PROGRAM StringHelper
VAR
END_VAR

METHOD EndsWith : BOOL
VAR_INPUT
	str		: Tc2_System.T_MaxString;
	char	: T_Char;	
END_VAR
EndsWith := Tc2_Standard.RIGHT(str, 1) = char;
END_METHOD

// Checks if the sourceString contains the stringToFind string. 
// Size of the source string is only limited to TwinCAT limitaitons, which in theory is not limited.
// Returns TRUE if found, else FALSE. Position of the found strimg is provided in the "position" output variable.
METHOD FindStringWithin : BOOL
VAR_INPUT
	sourceString	: ANY;	// String to look at
	stringToFind	: Tc2_System.T_MaxString; // String that should be containted in the sourceString
END_VAR
VAR_OUTPUT
	position	: DINT;	// Position of the found string
END_VAR

VAR
	tmpStr						: POINTER TO Tc2_System.T_MaxString;
	charIndex					: DINT;
	currentMatchingCharIndex	: DINT;
	tmpByte						: POINTER TO BYTE;
	firstCharPosition 			: dint;
END_VAR
IF NOT F_DoesVarTypeEqual(sourceString, IBaseLibrary.TYPE_STRING) THEN
	RETURN;
END_IF

IF sourceString.diSize <= SIZEOF(Tc2_System.T_MaxString) THEN
	tmpStr := __NEW(BYTE, SIZEOF(Tc2_System.T_MaxString));
	Tc2_System.MEMCPY(
		destAddr := tmpStr,
		srcAddr := sourceString.pValue,
		n := DINT_TO_UDINT(sourceString.diSize));
	//tmpStr := sourceString.pValue;
	position :=  Tc2_Standard.FIND(tmpStr^, stringToFind);
	FindStringWithin := position <> 0;
	__DELETE(tmpStr);
	RETURN;
END_IF

FOR charIndex := 0 TO sourceString.diSize BY 1 DO
	
	// Byte wise comparison, if matching byte, start filling the compared string
	tmpByte := sourceString.pValue + charIndex * SIZEOF(BYTE);
	// For debug purpose
	tmpStr := tmpByte;
	IF tmpbyte^ = stringToFind[currentMatchingCharIndex] THEN
		IF firstCharPosition = 0 THEN
			firstCharPosition := charIndex + 1;
		END_IF
		currentMatchingCharIndex := currentMatchingCharIndex + 1;
	ELSE
		currentMatchingCharIndex := 0;
		firstCharPosition := 0;
	END_IF
	
	// When index = str lenght - 1, we have found the entire string, exit the loop.
	IF currentMatchingCharIndex = (Tc2_Standard.LEN(stringToFind)) THEN
		position := firstCharPosition;
		FindStringWithin := TRUE;
		EXIT;
	END_IF
END_FOR
END_METHOD

// Joins the provided string with the string to add.
// The refStr is altered in the process, this no additional assignments are required as oposed to CONCAT which returns the resulting string.
METHOD Join
VAR_INPUT
	refStr		: REFERENCE TO Tc2_System.T_MaxString;
	strToJoin	: Tc2_System.T_MaxString;
END_VAR
refStr := Tc2_Standard.CONCAT(refStr, strToJoin);
END_METHOD

// Checks if STRING `str` starts with the `char`
// Returs TRUE if first character in the provided string is `char` provided
METHOD StartsWith : BOOL
VAR_INPUT
	str		: Tc2_System.T_MaxString;	// String to be checked
	char	: T_Char;	// Character that the string will be checked, if it starts with it.
END_VAR
StartsWith := Tc2_System.F_ToCHR(str[0]) = char;
END_METHOD

// Converts the provided string to all lower case and returns the converted value.
METHOD ToLowerCase : T_MaxString
VAR_INPUT
	str	: Tc2_System.T_MaxString;	// Source string
END_VAR
ToLowerCase := Tc2_Utilities.F_ToLCase(in := str);
END_METHOD

// Converts the input string to all lower case. Size of the string is irrelevant
METHOD ToLowerCase_UnlimitedSize
VAR_INPUT
	str	: ANY;
END_VAR

VAR
	charIndex	: DINT;
	ptrChar		: POINTER TO T_Char;
	char		: T_Char;
	malloc		: FB_Malloc(0,0);
	ptrByte		: POINTER TO BYTE;
END_VAR
IF NOT F_DoesVarTypeEqual(str, IBaseLibrary.TYPE_STRING) THEN
	RETURN;
END_IF

malloc.Allocate(1, str.diSize - 1);		
FOR charIndex := 0 TO str.diSize - 1 BY 1 DO
	ptrChar := str.pValue + DINT_TO_DWORD(charIndex);
	char := ToLowerCase(ptrChar^);
	ptrByte := ADR(char);
	malloc.Set(charIndex, ptrByte^);
END_FOR

Tc2_System.MEMCPY(
	destAddr := str.pValue, 
	srcAddr := malloc.Properties.StartAddress, 
	n := DINT_TO_UDINT(str.diSize - 1));
	
malloc.Free();
END_METHOD

// Converts the provided string to all upper case and returns the converted value.
METHOD ToUpperCase : Tc2_System.T_MaxString
VAR_INPUT
	str	: Tc2_System.T_MaxString;	// Source string
END_VAR
ToUpperCase := Tc2_Utilities.F_ToUCase(in := str);
END_METHOD

METHOD ToUpperCase_UnlimitedSize
VAR_INPUT
	str	: ANY;
END_VAR	

VAR
	charIndex	: DINT;
	ptrChar		: POINTER TO T_Char;
	char		: T_Char;
	malloc		: FB_Malloc(0,0);
	ptrByte		: POINTER TO BYTE;
END_VAR
IF NOT F_DoesVarTypeEqual(str, IBaseLibrary.TYPE_STRING) THEN
	RETURN;
END_IF

malloc.Allocate(1, str.diSize - 1);		
FOR charIndex := 0 TO str.diSize - 1 BY 1 DO
	ptrChar := str.pValue + DINT_TO_DWORD(charIndex);
	char := ToUpperCase(ptrChar^);
	ptrByte := ADR(char);
	malloc.Set(charIndex, ptrByte^);
END_FOR

Tc2_System.MEMCPY(
	destAddr := str.pValue, 
	srcAddr := malloc.Properties.StartAddress, 
	n := DINT_TO_UDINT(str.diSize - 1));
	
malloc.Free();
END_METHOD

// Removes leading spaces from the character string and returns the reduced character string
METHOD PUBLIC TrimLeftSide : Tc2_System.T_MaxString
VAR_INPUT
	str	: Tc2_System.T_MaxString; // String to be trimmed
END_VAR
TrimLeftSide := Tc2_Utilities.F_LTrim(in := str);
END_METHOD

// Truncates all trailing spaces from the specified value and returns the result.
METHOD PUBLIC TrimRightSide : Tc2_System.T_MaxString
VAR_INPUT
	str	: Tc2_System.T_MaxString;	// String to be trimmed
END_VAR
TrimRightSide := Tc2_Utilities.F_RTrim(in := str);
END_METHOD

END_PROGRAM

(* stored: Version 1.1.0.1, ProductVersion 3.1.4024.15
   POU StringHelper: Id {6038c506-8015-0cf2-2085-30a677155028}, SpecialFunc None
   Method EndsWith: Id {ae3c099d-30b2-0f82-0a20-ce3ad2e77fa0}
   Method FindStringWithin: Id {2f0f077d-67ad-00c3-05fa-2ccee8640db2}
   Method Join: Id {99346997-fd62-0afc-1ca1-062e8359a9d5}
   Method StartsWith: Id {5c75a7b6-3cc1-0540-0cd5-16739591bdb3}
   Method ToLowerCase: Id {04af86ff-c3c4-0ee5-29da-879b8d09b6b9}
   Method ToLowerCase_UnlimitedSize: Id {f4114202-5b66-0efa-14bc-fe041d3f54b7}
   Method ToUpperCase: Id {a9f90e08-f042-0b48-3d37-79d4dbe88971}
   Method ToUpperCase_UnlimitedSize: Id {3ed9e680-0d6f-0cbd-294a-745be70d999d}
   Method TrimLeftSide: Id {aaf318c8-56f7-0f39-3b6b-023f532313ad}
   Method TrimRightSide: Id {76095d0f-b051-05a8-3966-5a98e10f20ea} *)
